// TwinCAT 3 PLC project PLC_1
// ProgramVersion: 3.1.4024.0
// libraries:
//   Tc2_MC2, * (Beckhoff Automation GmbH)
//   Tc2_Standard, * (Beckhoff Automation GmbH)
//   Tc2_System, * (Beckhoff Automation GmbH)
//   Tc3_Module, * (Beckhoff Automation GmbH)
// project tree:
//   DUTs/ NcAxisRefStatus.TcDUT
//   / PlcTask.TcTTO
//   POUs/ MAIN.TcPOU
//   POUs/OOP/Axis Classes/ DCAxis.TcPOU, ParentAxis.TcPOU, ServoAxis.TcPOU, StepperAxis.TcPOU
//   POUs/OOP/Interfaces/ ITF_AxisControl.TcIO, ITF_CyclicUpdate.TcIO
//   POUs/OOP/State Managers/ AxisControlManager.TcPOU, StateProgram.TcPOU
//   Project Planning/ Class Diagram.TcCD (not stored)
// real-time tasks:
//   TASK PlcTask: cycle T#10ms, priority 20, ADS port 350
// motion (NC):
//   TASK NC-Task 1 SAF: cycle T#2ms, priority 4, ADS port 501
//   TASK NC-Task 1 SVB: cycle T#10ms, priority 8, ADS port 511
//   AXIS Stepper (id 1)
//     OtherSettings: AllowMotionCmdToSlave=true
//     encoder EncType=1
//     drive DrvType=5
//       Analog: TorqueSetpointScale=10, ScaleFactorActTorque=0.1
//       TimeComp: TaskDelayCycles=1
//     controller CtrType=1
//       CtrPara: PriorControlFactor=1
//         Observer: BandWidth=20
//   AXIS Servo (id 2)
//     OtherSettings: AllowMotionCmdToSlave=true
//     encoder EncType=1
//     drive DrvType=5
//       Analog: TorqueSetpointScale=10, ScaleFactorActTorque=0.1
//       TimeComp: TaskDelayCycles=1
//     controller CtrType=1
//       CtrPara: PriorControlFactor=1
//         Observer: BandWidth=20
//   AXIS DC (id 3)
//     OtherSettings: AllowMotionCmdToSlave=true
//     encoder EncType=1
//     drive DrvType=5
//       Analog: TorqueSetpointScale=10, ScaleFactorActTorque=0.1
//       TimeComp: TaskDelayCycles=1
//     controller CtrType=1
//       CtrPara: PriorControlFactor=1
//         Observer: BandWidth=20
// variable links:
//   PLC 1/PLC 1 Instance <-> NC-Task 1 SAF/Axes/Servo
//     PlcTask Inputs/StateProgram.Servo1._AxisReference.NcToPlc <-> Outputs/ToPlc
//     PlcTask Outputs/StateProgram.Servo1._AxisReference.PlcToNc <-> Inputs/FromPlc

CONFIGURATION PLC_1
    RESOURCE PLC ON TwinCAT3
        TASK PlcTask(INTERVAL := T#10ms, PRIORITY := 20);
        PROGRAM MAIN WITH PlcTask : MAIN;
    END_RESOURCE
END_CONFIGURATION

// ---- DUTs/NcAxisRefStatus.TcDUT
TYPE NcAxisRefStatus :
STRUCT
	
	_Error				: BOOL;
	_ErrorID			: UDINT;
	_ErrorStop			: BOOL;
	_Disabled			: BOOL;
	_Stopping			: BOOL;
	_StandStill			: BOOL;
	_DiscreteMotion		: BOOL;
	_ContinuousMotion	: BOOL;
	_SynchronizedMotion	: BOOL;
	_Homing				: BOOL;
	_ConstantVelocity	: BOOL;
	_Accelerating		: BOOL;
	_Decelerating		: BOOL;
	_Status				: ST_AxisStatus;
	
END_STRUCT
END_TYPE

// ---- POUs/OOP/Interfaces/ITF_AxisControl.TcIO
INTERFACE ITF_AxisControl

METHOD StartDisable : BOOL
VAR_INPUT
END_VAR
END_METHOD

METHOD StartEnable : BOOL
VAR_INPUT
END_VAR
END_METHOD

METHOD StartErrorChecking : BOOL
VAR_INPUT
END_VAR
END_METHOD

METHOD StartMovement : BOOL
VAR_INPUT
END_VAR
END_METHOD

METHOD StartReset : BOOL
VAR_INPUT
END_VAR
END_METHOD

END_INTERFACE

// ---- POUs/OOP/Interfaces/ITF_CyclicUpdate.TcIO
INTERFACE ITF_CyclicUpdate

// Uses HRESULT outputs for management of different scenarios, such as errors and non-completes

//    0 - No Output / Execute In Progress
//    1 - Execute Complete
//    2 - Execute Failed, No Program Error, Object's Internal Timer Exceeded Limit.
//   -1 - Execute Failed, Program Error

METHOD CyclicUpdate : HRESULT

// Uses HRESULT outputs for management of different scenarios, such as errors and non-completes

//    0 - No Output / Execute In Progress
//    1 - Execute Complete
//    2 - Execute Failed, No Program Error, Object's Internal Timer Exceeded Limit.
//   -1 - Execute Failed, Program Error
END_METHOD

END_INTERFACE

// ---- POUs/MAIN.TcPOU
PROGRAM MAIN
VAR	
END_VAR

StateProgram();

END_PROGRAM

// ---- POUs/OOP/State Managers/StateProgram.TcPOU
PROGRAM StateProgram
VAR
	
	Stepper1				: StepperAxis;
	Servo1					: ServoAxis;
	DC1						: DCAxis;
	AxisControlManager		: AxisControlManager;
	
	iAxesManagerCycle		: ITF_CyclicUpdate := AxisControlManager;
	iAxesIndividualCycle	: ARRAY [0..2] OF ITF_CyclicUpdate := [Stepper1, Servo1, DC1];
	
	Result					: HRESULT;
	i						: INT;
	State					: INT;
	
END_VAR


// Switch between the targetted axes AFTER axis functionality has finished
// Prevents switching mid-movement

FOR i := 0 TO 1 BY 1 DO
	iAxesIndividualCycle[i].CyclicUpdate();
END_FOR

Result := iAxesManagerCycle.CyclicUpdate();

CASE State OF
	
	0:
		State := 0;
	
	1:
		AxisControlManager.TargetAxis := Stepper1;
		IF Result = 1 THEN
			State := 0;
		END_IF
		
	2:
		AxisControlManager.TargetAxis := Servo1;
		IF Result = 1 THEN
			State := 0;
		END_IF
		
	3:
		AxisControlManager.TargetAxis := DC1;
		IF Result = 1 THEN
			State := 0;
		END_IF
	
END_CASE

END_PROGRAM

// ---- POUs/OOP/Axis Classes/StepperAxis.TcPOU
FUNCTION_BLOCK StepperAxis EXTENDS ParentAxis
VAR
END_VAR

METHOD StartDisable : BOOL
StartDisable := TRUE;
RETURN;
END_METHOD

METHOD StartEnable : BOOL
StartEnable := TRUE;
RETURN;
END_METHOD

METHOD StartErrorChecking : BOOL
StartErrorChecking := TRUE;
RETURN;
END_METHOD

METHOD StartMovement : BOOL
StartMovement := TRUE;
RETURN;
END_METHOD

METHOD StartReset : BOOL
StartReset := TRUE;
RETURN;
END_METHOD

END_FUNCTION_BLOCK

// ---- POUs/OOP/Axis Classes/ParentAxis.TcPOU
{attribute 'no_explicit_call' := 'Do not call this POU directly'}
FUNCTION_BLOCK ParentAxis IMPLEMENTS ITF_AxisControl, ITF_CyclicUpdate
VAR
	
	// DO NOT USE DIRECTLY 
	// THIS IS A PARENT CLASS DESIGNED TO PROVIDE A BASE OF KEY VARIABLES / METHODS FOR SUB AXIS CLASSES
	
	_ClassRunningIndicatorToggle	: BOOL;
	
	_LocalState						: INT := 0;
	_InternalCounter				: INT := 0;
	_i								: INT := 0;
	_ErrorCount						: UDINT := 0;
	_CurrentErrorCode				: UDINT := 0;
	_PreviousErrorCode				: UDINT := 0;
	
	
	_IsBusyMoving					: BOOL := FALSE;
	_IsBusyStopping					: BOOL := FALSE;
	_IsReadyForCommand				: BOOL := FALSE;
	_IsDoneWithCommand				: BOOL := FALSE;
	_IsInError						: BOOL := FALSE;
	
	_ErrorRTrig						: R_TRIG;
	
END_VAR

// DO NOT USE DIRECTLY 
// THIS IS A PARENT CLASS DESIGNED TO PROVIDE A BASE OF KEY VARIABLES / METHODS FOR SUB AXIS CLASSES

{attribute 'no_explicit_call' := 'Do not call this METHOD directly'}
METHOD CyclicUpdate : HRESULT
VAR_INPUT
END_VAR
END_METHOD

{attribute 'no_explicit_call' := 'Do not call this METHOD directly'}
METHOD StartDisable : BOOL
StartDisable := TRUE;
RETURN;
END_METHOD

{attribute 'no_explicit_call' := 'Do not call this METHOD directly'}
METHOD StartEnable : BOOL
StartEnable := TRUE;
RETURN;
END_METHOD

{attribute 'no_explicit_call' := 'Do not call this METHOD directly'}
METHOD StartErrorChecking : BOOL
StartErrorChecking := TRUE;
RETURN;
END_METHOD

{attribute 'no_explicit_call' := 'Do not call this METHOD directly'}
METHOD StartMovement : BOOL
StartMovement := TRUE;
RETURN;
END_METHOD

{attribute 'no_explicit_call' := 'Do not call this METHOD directly'}
METHOD StartReset : BOOL
StartReset := TRUE;
RETURN;
END_METHOD

END_FUNCTION_BLOCK

// ---- POUs/OOP/Axis Classes/ServoAxis.TcPOU
FUNCTION_BLOCK ServoAxis EXTENDS ParentAxis
VAR
	
	_AxisReference				: AXIS_REF;
	
	_Enable						: MC_Power;
	_ReadStatus					: MC_ReadStatus;
	_Reset						: MC_Reset;
	_MoveRelative				: MC_MoveRelative;
	
	_Status						: NcAxisRefStatus;
	
END_VAR

METHOD CyclicUpdate : HRESULT
VAR_INPUT
END_VAR

_ClassRunningIndicatorToggle := NOT(_ClassRunningIndicatorToggle);

_Enable(Axis := _AxisReference);
_Reset(Axis := _AxisReference);
_MoveRelative(Axis := _AxisReference);

_ReadStatus
(
	Axis 					:= _AxisReference,
	Enable 					:= TRUE,
	Error 					=> _Status._Error,
	ErrorID 				=> _Status._ErrorID,
	ErrorStop 				=> _Status._ErrorStop,
	Disabled 				=> _Status._Disabled,
	Stopping 				=> _Status._Stopping,
	StandStill 				=> _Status._StandStill,
	DiscreteMotion 			=> _Status._DiscreteMotion,
	ContinuousMotion 		=> _Status._ContinuousMotion,
	SynchronizedMotion 		=> _Status._SynchronizedMotion,
	Homing 					=> _Status._Homing,
	ConstantVelocity 		=> _Status._ConstantVelocity,
	Accelerating 			=> _Status._Accelerating,
	Decelerating 			=> _Status._Decelerating,
	Status 					=> _Status._Status
);

_IsBusyMoving :=
(
	_ReadStatus.DiscreteMotion OR
	_ReadStatus.ConstantVelocity OR
	_ReadStatus.SynchronizedMotion
);

_IsBusyStopping :=
(
	_ReadStatus.Stopping
);

_IsReadyForCommand :=
(
	NOT(_ReadStatus.Disabled) AND
	NOT(_IsBusyMoving) AND
	NOT(_IsBusyStopping) AND
	NOT(_ReadStatus.Error) AND
	NOT(_ReadStatus.ErrorStop)
);

_IsDoneWithCommand :=
(
	_Reset.Done OR
	_MoveRelative.Done
);

_IsInError :=
(
	_ReadStatus.Error
);

_CurrentErrorCode := _ReadStatus.ErrorID;
	
IF _Status._ErrorID <> 0 THEN
	_PreviousErrorCode := _ReadStatus.ErrorID;
END_IF

_ErrorRTrig(CLK := _IsInError);
IF _ErrorRTrig.Q THEN
	_ErrorCount := _ErrorCount + 1;
END_IF


CyclicUpdate := 1;
RETURN;
END_METHOD

METHOD StartDisable : BOOL
_Enable(Axis := _AxisReference);

_Enable.Enable := FALSE;
_Enable.Enable_Negative := FALSE;
_Enable.Enable_Positive := FALSE;
_Enable.Override := 0;

IF NOT(_Enable.Status) THEN
	StartDisable := TRUE;
	RETURN;
ELSE
	;
END_IF

RETURN;
END_METHOD

METHOD StartEnable : BOOL
_Enable(Axis := _AxisReference);

_Enable.Enable := TRUE;
_Enable.Enable_Negative := TRUE;
_Enable.Enable_Positive := TRUE;
_Enable.Override := 100;

IF _Enable.Error THEN
	_Enable.Enable := FALSE;
	StartEnable := FALSE;
	RETURN;
ELSE
	;
END_IF

IF _Enable.Status THEN
	StartEnable := TRUE;
	RETURN;
ELSE
	;
END_IF

RETURN;
END_METHOD

METHOD StartErrorChecking : BOOL
IF _IsInError THEN
	StartErrorChecking := TRUE;
	RETURN;
ELSE
	;
END_IF

RETURN;
END_METHOD

METHOD StartMovement : BOOL
_MoveRelative(Axis := _AxisReference);
_MoveRelative.Distance := 100;
_MoveRelative.Velocity := 20;
_MoveRelative.Execute := TRUE;

IF _MoveRelative.Error THEN
	_MoveRelative.Execute := FALSE;
	StartMovement := FALSE;
	RETURN;
ELSE
	;
END_IF

IF _MoveRelative.Done THEN
	_MoveRelative.Execute := FALSE;
	StartMovement := TRUE;
	RETURN;
ELSE
	;
END_IF

RETURN;
END_METHOD

METHOD StartReset : BOOL
_MoveRelative(Axis := _AxisReference);
_Reset(Axis := _AxisReference);

_MoveRelative.Execute := FALSE;

_Reset.Execute := TRUE;

IF _Reset.Error THEN
	_Reset.Execute := FALSE;
	StartReset := FALSE;
	RETURN;
ELSE
	;
END_IF

IF _Reset.Done THEN
	_Reset.Execute := FALSE;
	StartReset := TRUE;
ELSE
	;
END_IF
END_METHOD

END_FUNCTION_BLOCK

// ---- POUs/OOP/Axis Classes/DCAxis.TcPOU
FUNCTION_BLOCK DCAxis EXTENDS ParentAxis
VAR
END_VAR

METHOD StartDisable : BOOL
StartDisable := TRUE;
RETURN;
END_METHOD

METHOD StartEnable : BOOL
StartEnable := TRUE;
RETURN;
END_METHOD

METHOD StartErrorChecking : BOOL
StartErrorChecking := TRUE;
RETURN;
END_METHOD

METHOD StartMovement : BOOL
StartMovement := TRUE;
RETURN;
END_METHOD

METHOD StartReset : BOOL
StartReset := TRUE;
RETURN;
END_METHOD

END_FUNCTION_BLOCK

// ---- POUs/OOP/State Managers/AxisControlManager.TcPOU
FUNCTION_BLOCK AxisControlManager IMPLEMENTS ITF_CyclicUpdate
VAR
	
	// State machine for simple axis movement
	// Aims to turn on an axis, command it do do a movement, then disable it
	// Highest level state machine
	// Call METHOD to run, call PROPERTY to switch axis
	
	_AxisControl			: ITF_AxisControl;
	
	_LocalState				: INT;
	
END_VAR

METHOD CyclicUpdate : HRESULT

// If interface has not been assigned, exit method
IF _AxisControl = 0 THEN
	CyclicUpdate := 0;
	RETURN;
END_IF

IF _AxisControl.StartErrorChecking() THEN
	_LocalState := 99;
END_IF

// Turn axis on, execute its movement, turn axis off
CASE _LocalState OF
	
	0:
		_LocalState := 1;
		
	1:
		IF _AxisControl.StartEnable() THEN
			_LocalState := 2;
		END_IF
		
	2:
		IF _AxisControl.StartMovement() THEN
			_LocalState := 3;
		END_IF
		
	3:
		IF _AxisControl.StartDisable() THEN
			_LocalState := 4;
		END_IF
		
	4:
		_LocalState := 4;
		CyclicUpdate := 1;
		RETURN;
		
	99:
		IF _AxisControl.StartReset() THEN
			_LocalState := 0;
		END_IF
	
END_CASE
END_METHOD

PROPERTY TargetAxis : ITF_AxisControl
GET
TargetAxis := _AxisControl;
END_GET
SET
_AxisControl := TargetAxis;
END_SET
END_PROPERTY

END_FUNCTION_BLOCK
